// LS Electric XG5000 project: gh
// PLC LSPLC
// module base 0 slot 0: 입출력 모듈:XBC-DR32H (DC 24V 입력, 릴레이 출력 32점)
// module base 0 slot 1: 위치결정 모듈:XBF-PD02A (위치결정 펄스(LD)출력형, 2축)
// module base 0 slot 2: 출력 모듈:XBE-TN/TP16A (트랜지스터 출력, 16점 (싱크출력/소스출력))

PROGRAM NewProgram (task: 스캔 프로그램)

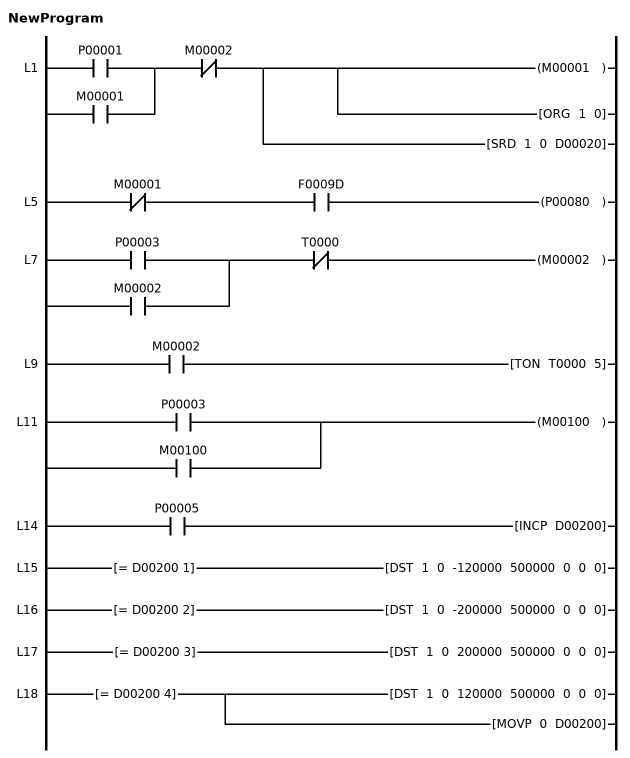
; L1
LOAD      P00001
OR        M00001
AND NOT   M00002
OUT       M00001
ORG       1 0
SRD       1 0 D00020
; L5
LOAD NOT  M00001
AND       F0009D
OUT       P00080
; L7
LOAD      P00003
OR        M00002
AND NOT   T0000
OUT       M00002
; L9
LOAD      M00002
TON       T0000 5
; L11
LOAD      P00003
OR        M00100
OUT       M00100
; L14
LOAD      P00005
INCP      D00200
; L15
LOAD=     D00200 1
DST       1 0 -120000 500000 0 0 0
; L16
LOAD=     D00200 2
DST       1 0 -200000 500000 0 0 0
; L17
LOAD=     D00200 3
DST       1 0 200000 500000 0 0 0
; L18
LOAD=     D00200 4
DST       1 0 120000 500000 0 0 0
MOVP      0 D00200